Fanuc KAREL source: port_OPIN.kl

PROGRAM TP
%NOLOCKGROUP
VAR
 x: BOOLEAN
BEGIN
 x = OPIN[3]
END TP
